// TwinCAT 3 PLC project Untitled1
// ProgramVersion: 3.1.4024.0
// libraries:
//   Tc2_Standard, * (Beckhoff Automation GmbH)
//   Tc2_System, * (Beckhoff Automation GmbH)
//   Tc3_Module, * (Beckhoff Automation GmbH)
// project tree:
//   DUTs/ KOMANDA.TcDUT, POZAYZ.TcDUT, POZICIJA.TcDUT, Valj.TcDUT
//   GVLs/ AUTO.TcGVL, GVL.TcGVL
//   / PlcTask.TcTTO
//   POUs/ AutoMove.TcPOU, Counter.TcPOU, Init.TcPOU, MAIN.TcPOU, Motor.TcPOU, MotorControla.TcPOU, Multiplex.TcPOU, Automatic.TcPOU, AutoMove2.TcPOU, Motor2.TcPOU, Test.TcPOU, TrackingLogic.TcPOU

CONFIGURATION Untitled1
    RESOURCE PLC ON TwinCAT3
        TASK PlcTask(INTERVAL := T#10ms, PRIORITY := 20);
        PROGRAM Automatic WITH PlcTask : Automatic;
    END_RESOURCE
END_CONFIGURATION

// ---- DUTs/KOMANDA.TcDUT
TYPE KOMANDA :
STRUCT
	I: INT;
	T: INT;
	P : INT;
END_STRUCT
END_TYPE

// ---- DUTs/POZAYZ.TcDUT
TYPE POZAYZ :
STRUCT
	A: INT;
	Y: INT;
	Z: INT;
END_STRUCT
END_TYPE

// ---- DUTs/POZICIJA.TcDUT
TYPE POZICIJA :
STRUCT
	A: INT;
	Y: INT;
	Z: INT;
	P: INT;
END_STRUCT
END_TYPE

// ---- DUTs/Valj.TcDUT
TYPE Valj :
STRUCT
	id: INT;
	pos: POZICIJA;
END_STRUCT
END_TYPE

// ---- GVLs/AUTO.TcGVL
{attribute 'qualified_only'}
VAR_GLOBAL
	Init : BOOL := FALSE;
	Varno :BOOL := FALSE;
	MotorIzbira : INT;
	VrtenjePremik : BOOL;
	VrtenjeSmer : BOOL;
	DvigPremik : BOOL;
	DvigSmer : BOOL;
	IztegPremik : BOOL;
	IztegSmer : BOOL;
	PrijemPremik : BOOL;
	PrijemSmer : BOOL;
	Current: POZICIJA;
	N: INT := 5; //v InstructionSize
	Komande0: ARRAY [0..4] OF POZICIJA := [(A := 0, Y := 0, Z := 0, P:= 0 ), 
		(A := 100, Y := 40, Z := 50, P:= 15 ),
		(A := 80, Y := 20, Z := 30, P:= 0 ),
		(A := 120, Y := 0, Z := 15, P:= 12 ),
		(A := 100, Y := 0, Z := 15, P:= 0 )];
	Status: INT := 0;
	PositionNum: INT := 2; // ne rabi
	ItemNumber : INT := 2; //ne rabi
	StageSelect : INT := 0;
	Recept : INT := 0;
	VRoki : INT := 0;
	Prijem : BOOL := FALSE;
	Positions: ARRAY [1..11] OF POZAYZ := [
			(A := 30, Y:=60, Z:= 105),
			(A := 30, Y:=60, Z:= 62),
			(A := 30, Y:=60, Z:= 20),
			(A := 60, Y:=60, Z:= 105),
			(A := 60, Y:=60, Z:= 62), // 5
			(A := 50, Y:=60, Z:= 105),
			(A := 50, Y:=60, Z:= 62),
			(A := 37, Y:=60, Z:= 105),
			(A := 40, Y:=45, Z:= 105),
			(A := 47, Y:=60, Z:= 105), // 10
			(A := 33, Y:=0, Z:= 50)];
	Items: ARRAY [1..5] OF POZAYZ := [
			(A := 5, Y:=60, Z:= 20),
			(A := 5, Y:=60, Z:= 62),
			(A := 5, Y:=60, Z:= 105),
			(A := 50, Y:=60, Z:= 105),
			(A := 50, Y:=60, Z:= 62)];
	StageMax : INT :=10;
	Stages :  ARRAY [1 .. 3] OF ARRAY [1 .. 9] OF KOMANDA :=  [[
		(I := 1, T := 0, P := 16),
		(I := 0, T := 1, P := 0),
		(I := 2, T := 0, P := 16),
		(I := 0, T := 2, P := 0),
		(I := 3, T := 0, P := 16), // 5
		(I := 0, T := 3, P := 0),
		(I := 2, T := 0, P := 16),
		(I := 0, T := 9, P := 0),
		(I := 0, T := 11, P := 0)],
[
		(I := 5, T := 0, P := 16),
		(I := 0, T := 4, P := 0),
		(I := 4, T := 0, P := 16),
		(I := 0, T := 5, P := 0),
		(I := 4, T := 0, P := 16), // 5
		(I := 0, T := 6, P := 0),
		(I := 5, T := 0, P := 16),
		(I := 0, T := 7, P := 0),
		(I := 0, T := 11, P := 0)],
[
		(I := 1, T := 0, P := 16),
		(I := 0, T := 10, P := 0),
		(I := 2, T := 0, P := 16),
		(I := 0, T := 8, P := 0),
		(I := 3, T := 0, P := 16), // 5
		(I := 0, T := 9, P := 0),
		(I := 3, T := 0, P := 16),
		(I := 0, T := 1, P := 0),
		(I := 0, T := 11, P := 0)]];
END_VAR

// ---- GVLs/GVL.TcGVL
{attribute 'Iualified_only'}


VAR_GLOBAL
	ToggleSwitch AT %I* : BOOL;
	LEDRed AT %Q* : BOOL;
	LEDGreen AT %Q* : BOOL;
	LEDUBlue AT %Q* : BOOL;
	LEDLBlue AT %Q* : BOOL;
	RedButton AT %I* : BOOL;
	GreenButton AT %I* : BOOL;
	ULBButton AT %I* : BOOL;
	URBButton AT %I* : BOOL;
	LLBButton AT %I* : BOOL;
	LRBButton AT %I* : BOOL;
	
	MVS AT %Q* : BOOL;
	MVP AT %Q* : BOOL;
	MIS AT %Q* : BOOL;
	MIP AT %Q* : BOOL;
	MDS AT %Q* : BOOL;
	MDP AT %Q* : BOOL;
	MPS AT %Q* : BOOL;
	MPP AT %Q* : BOOL;
	
	KSV AT %I* : BOOL;
	KSI AT %I* : BOOL;
	KSD AT %I* : BOOL;
	KSP AT %I* : BOOL;
	StV AT %I* : BOOL;
	StD AT %I* : BOOL;
	StI AT %I* : BOOL;
	StP AT %I* : BOOL;
END_VAR

// ---- POUs/Automatic.TcPOU
PROGRAM Automatic
VAR
	foo : BOOL;
	motor_1 : Motor2;
	auto_move : AutoMove;
	auto_move_2 : AutoMove2;
	tracking : TrackingLogic;
	init : Init;
END_VAR


init();
auto_move_2();
motor_1();
tracking();

END_PROGRAM

// ---- POUs/Motor2.TcPOU
FUNCTION_BLOCK Motor2
VAR_INPUT
END_VAR
VAR_OUTPUT
END_VAR
VAR
	sel1: BOOL := FALSE;
	sel2: BOOL := FALSE;
	sel3: BOOL := FALSE;
	sel4: BOOL := FALSE;
	mc1: motorControla;
	mc2: motorControla;
	mc3: motorControla;
	mc4: motorControla;
	interlock: BOOL;
	stop: BOOL;
END_VAR

IF GVL.ToggleSwitch = TRUE THEN
	AUTO.Varno := FALSE;
	IF GVL.ULBButton THEN
		sel1 := TRUE;
		sel2 := FALSE;
		sel3 := FALSE;
		sel4 := FALSE;
	ELSIF GVL.URBButton THEN
		sel1 := FALSE;
		sel2 := TRUE;
		sel3 := FALSE;
		sel4 := FALSE;
	ELSIF GVL.LLBButton THEN
		sel1 := FALSE;
		sel2 := FALSE;
		sel3 := TRUE;
		sel4 := FALSE;
	ELSIF GVL.LRBButton THEN
		sel1 := FALSE;
		sel2 := FALSE;
		sel3 := FALSE;
		sel4 := TRUE;
	END_IF
	
	mc1(		Premik := GVL.RedButton,
			Smer := GVL.GreenButton AND sel1,
			Select := sel1,
			KS := GVL.KSV,
			Step :=GVL.StV,
			Limes := 185,
			Position => AUTO.Current.A,
			OutSmer => GVL.MVS,
			OutPremik => GVL.MVP,
			Interlock => interlock,
			Stop => stop
			);
mc2(		Premik := GVL.RedButton,
			Smer := GVL.GreenButton AND sel2,
			Select := sel2,
			KS := GVL.KSD,
			Step :=GVL.StD,
			Limes := 105,
			Position => AUTO.Current.Z,
			OutSmer => GVL.MDS,
			OutPremik => GVL.MDP,
			Interlock => interlock,
			Stop => stop);
		mc3(
			Premik := GVL.RedButton,
			Smer := GVL.GreenButton AND sel3,
			Select := sel3,
			KS := GVL.KSI,
			Step :=GVL.StI,
			Limes := 65,
			Position => AUTO.Current.Y,
			OutSmer => GVL.MIS,
			OutPremik => GVL.MIP,
			Interlock => interlock,
			Stop => stop);
		mc4(
			Premik := GVL.RedButton,
			Smer := GVL.GreenButton AND sel4,
			Select := sel4,
			KS := GVL.KSP,
			Step :=GVL.StP,
			Limes := 16,
			Position => AUTO.Current.P,
			OutSmer => GVL.MPS,
			OutPremik => GVL.MPP,
			Interlock => interlock,
			Stop => stop);
ELSE
	CASE AUTO.MotorIzbira OF
		1:
		sel1 := TRUE;
		sel2 := FALSE;
		sel3 := FALSE;
		sel4 := FALSE;
	2:
		sel1 := FALSE;
		sel2 := TRUE;
		sel3 := FALSE;
		sel4 := FALSE;
	3:
		sel1 := FALSE;
		sel2 := FALSE;
		sel3 := TRUE;
		sel4 := FALSE;
	4:
		sel1 := FALSE;
		sel2 := FALSE;
		sel3 := FALSE;
		sel4 := TRUE;
	END_CASE
		mc1(
			Premik := AUTO.VrtenjePremik,
			Smer := AUTO.VrtenjeSmer,
			Select := sel1,
			KS := GVL.KSV,
			Step :=GVL.StV,
			Limes := 185,
			Position => AUTO.Current.A,
			OutPremik => GVL.MVP,
			OutSmer => GVL.MVS,
			Interlock => interlock,
			Stop => stop
			);
		mc2(
			Premik := AUTO.DvigPremik,
			Smer := AUTO.DvigSmer,
			Select := sel2,
			KS := GVL.KSD,
			Step :=GVL.StD,
			Limes := 105,
			Position => AUTO.Current.Z,
			OutPremik => GVL.MDP,
			OutSmer => GVL.MDS,
			Interlock => interlock,
			Stop => stop
			);
		
		IF AUTO.Current.Y = 0 AND AUTO.IztegSmer = TRUE THEN
			//GVL.LEDLBlue := TRUE;
			ELSE
			//.LEDLBlue := FALSE;
			mc3(
			Premik := AUTO.IztegPremik,
			Smer := AUTO.IztegSmer,
			Select := sel3,
			KS := GVL.KSI,
			Step :=GVL.StI,
			Limes := 60,
			Position => AUTO.Current.Y,
			OutPremik => GVL.MIP,
			OutSmer => GVL.MIS,
			Interlock => interlock,
			Stop => stop
			);
			END_IF
		mc4(
			Premik := AUTO.PrijemPremik,
			Smer := AUTO.PrijemSmer,
			Select := sel4,
			KS := GVL.KSP,
			Step :=GVL.StP,
			Limes := 16,
			Position => AUTO.Current.P,
			OutPremik => GVL.MPP,
			OutSmer => GVL.MPS,
			Interlock => interlock,
			Stop => stop
			);
END_IF

GVL.LEDGreen := stop;
GVL.LEDRed := interlock;

RETURN;

END_FUNCTION_BLOCK

// ---- POUs/MotorControla.TcPOU
FUNCTION_BLOCK MotorControla
VAR_INPUT
	Premik: BOOL;
	Smer: BOOL;
	Select: BOOL;
	KS: BOOL;
	Step: BOOL;
	Limes: WORD;
END_VAR
VAR_OUTPUT
	OutPremik: BOOL;
	OutSmer: BOOL;
	Interlock: BOOL;
	Stop: BOOL;
	Position: WORD;
END_VAR
VAR
	R_TRIG_0: R_TRIG;
	Dump: TIME;
	InL: TOF;
	RS_0: RS;

	R_TRIG_1: R_TRIG;
	TON0: TON;
	TON1: TON;
	TON_0: TON;
	Counter_0: Counter;
	F_TRIG_0: F_TRIG;
	InL1: TOF;
	IntL1: BOOL;
	IntL2: BOOL;
	IntL3: BOOL;
	R_TRIG_2: R_TRIG;
END_VAR
//dODAJ COLLISION DETECTION AND AVOIDANCE
//ZRIHTAJ SMER, KI SE SLABO SPREMINJA

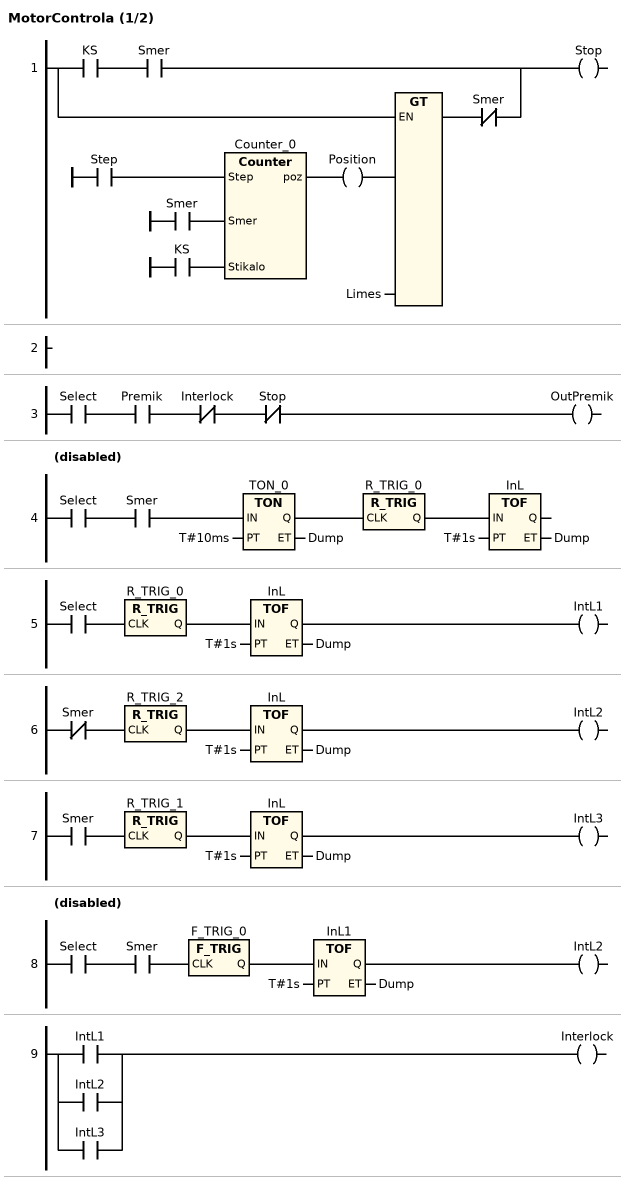
// NETWORK 1
Counter_0(Step := Step, Smer := Smer, Stikalo := KS); // Counter
Position := Counter_0.poz;
Stop := KS AND Smer OR Counter_0.poz > Limes AND NOT Smer;

// NETWORK 2

// NETWORK 3
OutPremik := Select AND Premik AND NOT Interlock AND NOT Stop;

// NETWORK 4 (disabled)
// TON_0(IN := Select AND Smer, PT := T#10ms, ET => Dump); // TON
// R_TRIG_0(CLK := TON_0.Q); // R_TRIG
// InL(IN := R_TRIG_0.Q, PT := T#1s, ET => Dump); // TOF

// NETWORK 5
R_TRIG_0(CLK := Select); // R_TRIG
InL(IN := R_TRIG_0.Q, PT := T#1s, ET => Dump); // TOF
IntL1 := InL.Q;

// NETWORK 6
R_TRIG_2(CLK := NOT Smer); // R_TRIG
InL(IN := R_TRIG_2.Q, PT := T#1s, ET => Dump); // TOF
IntL2 := InL.Q;

// NETWORK 7
R_TRIG_1(CLK := Smer); // R_TRIG
InL(IN := R_TRIG_1.Q, PT := T#1s, ET => Dump); // TOF
IntL3 := InL.Q;

// NETWORK 8 (disabled)
// F_TRIG_0(CLK := Select AND Smer); // F_TRIG
// InL1(IN := F_TRIG_0.Q, PT := T#1s, ET => Dump); // TOF
// IntL2 := InL1.Q;

// NETWORK 9
Interlock := IntL1 OR IntL2 OR IntL3;

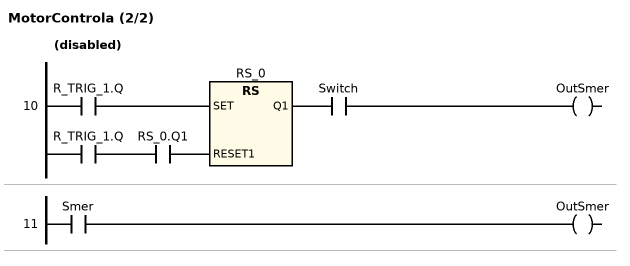
// NETWORK 10 (disabled)
// RS_0(SET := R_TRIG_1.Q, RESET1 := R_TRIG_1.Q AND RS_0.Q1); // RS
// OutSmer := RS_0.Q1 AND Switch;

// NETWORK 11
OutSmer := Smer;

END_FUNCTION_BLOCK

// ---- POUs/Counter.TcPOU
FUNCTION_BLOCK Counter
VAR_INPUT
	Step: BOOL;
	Smer: BOOL;
	Stikalo: BOOL;
END_VAR
VAR_OUTPUT
	poz: WORD;
END_VAR
VAR
	R_TRIG_0: R_TRIG;
	CTUD_0: Tc2_Standard.CTUD;
	R_TRIG_1: Tc2_Standard.R_TRIG;
END_VAR

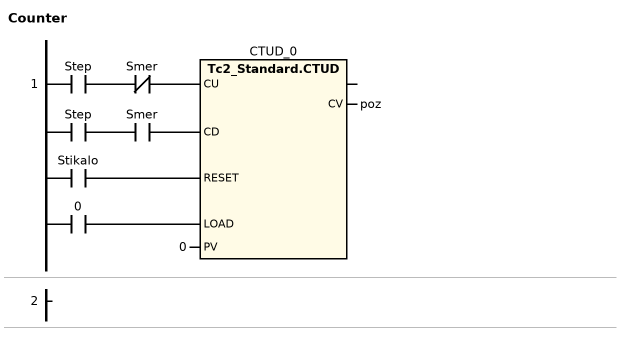
// NETWORK 1
CTUD_0(CU := Step AND NOT Smer, CD := Step AND Smer, RESET := Stikalo, LOAD := 0, PV := 0, CV => poz); // Tc2_Standard.CTUD

// NETWORK 2

END_FUNCTION_BLOCK

// ---- POUs/AutoMove.TcPOU
FUNCTION_BLOCK AutoMove
VAR_INPUT
END_VAR
VAR_OUTPUT
END_VAR
VAR
END_VAR

IF AUTO.Status > 0 AND AUTO.Status < AUTO.N THEN
	IF AUTO.Current.A <> AUTO.Komande0[AUTO.Status].A  THEN
		AUTO.MotorIzbira := 1;
		IF AUTO.Current.A > AUTO.Komande0[AUTO.Status].A THEN
			AUTO.VrtenjeSmer := TRUE;
		ELSE
			AUTO.VrtenjeSmer := FALSE;
		END_IF
		AUTO.VrtenjePremik := TRUE;
	ELSIF AUTO.Current.Y <> AUTO.Komande0[AUTO.Status].Y  THEN
		AUTO.MotorIzbira := 3;
		IF AUTO.Current.Y > AUTO.Komande0[AUTO.Status].Y THEN
			AUTO.IztegSmer := TRUE;
		ELSE
			AUTO.IztegSmer := FALSE;
		END_IF
		AUTO.IztegPremik := TRUE;
	ELSIF AUTO.Current.Z <> AUTO.Komande0[AUTO.Status].Z  THEN
		AUTO.MotorIzbira := 2;
		IF AUTO.Current.Z > AUTO.Komande0[AUTO.Status].Z THEN
			AUTO.DvigSmer := TRUE;
		ELSE
			AUTO.DvigSmer := FALSE;
		END_IF
		AUTO.DvigPremik := TRUE;
	ELSIF AUTO.Current.P <> AUTO.Komande0[AUTO.Status].P  THEN
		AUTO.MotorIzbira := 4;
		IF AUTO.Current.P > AUTO.Komande0[AUTO.Status].P THEN
			AUTO.PrijemSmer := TRUE;
		ELSE
			AUTO.PrijemSmer := FALSE;
		END_IF
		AUTO.PrijemPremik := TRUE;
	ELSE
		AUTO.VrtenjePremik := FALSE;
		AUTO.DvigPremik := FALSE;
		AUTO.IztegPremik := FALSE;
		AUTO.PrijemPremik := FALSE;
		AUTO.Status := AUTO.Status + 1;
	END_IF
END_IF

END_FUNCTION_BLOCK

// ---- POUs/AutoMove2.TcPOU
FUNCTION_BLOCK AutoMove2
VAR_INPUT
END_VAR
VAR_OUTPUT
END_VAR
VAR
	Target : POZAYZ;
END_VAR

IF AUTO.Init AND AUTO.StageSelect > 0 AND AUTO.StageSelect < AUTO.StageMax THEN
	IF AUTO.Varno = FALSE THEN
		AUTO.MotorIzbira := 3;
		AUTO.IztegSmer := TRUE;
		AUTO.IztegPremik := TRUE;
		IF AUTO.Current.Y = 0 THEN
			AUTO.Varno := TRUE;
		END_IF
	ELSIF AUTO.Stages[AUTO.Recept][Auto.StageSelect].I = 0 THEN
		Target := AUTO.Positions[AUTO.Stages[AUTO.Recept][Auto.StageSelect].T];
		IF AUTO.Current.Z <> Target.Z  THEN
			AUTO.MotorIzbira := 2;
			IF AUTO.Current.Z > Target.Z THEN
				AUTO.DvigSmer := TRUE;
			ELSE
				AUTO.DvigSmer := FALSE;
			END_IF
		AUTO.DvigPremik := TRUE;
		ELSIF AUTO.Current.A <> Target.A  THEN
			AUTO.MotorIzbira := 1;
			IF AUTO.Current.A > Target.A THEN
				AUTO.VrtenjeSmer := TRUE;
			ELSE
				AUTO.VrtenjeSmer := FALSE;
			END_IF
			AUTO.VrtenjePremik := TRUE;
		ELSIF AUTO.Current.Y <> Target.Y  THEN
			AUTO.MotorIzbira := 3;
			IF AUTO.Current.Y > Target.Y THEN
				AUTO.IztegSmer := TRUE;
			ELSE
				AUTO.IztegSmer := FALSE;
			END_IF
			AUTO.IztegPremik := TRUE;
		ELSIF AUTO.Current.P <> AUTO.Stages[AUTO.Recept][Auto.StageSelect].P  THEN
			AUTO.MotorIzbira := 4;
			IF AUTO.Current.P > AUTO.Stages[AUTO.Recept][Auto.StageSelect].P THEN
				AUTO.PrijemSmer := TRUE;
			ELSE
				AUTO.PrijemSmer := FALSE;
			END_IF
			AUTO.PrijemPremik := TRUE;
		ELSE
			AUTO.VrtenjePremik := FALSE;
			AUTO.DvigPremik := FALSE;
			AUTO.IztegPremik := FALSE;
			AUTO.PrijemPremik := FALSE;
			AUTO.StageSelect := AUTO.StageSelect + 1;
			AUTO.Varno := FALSE;
		END_IF
	ELSE
		Target := AUTO.Items[AUTO.Stages[AUTO.Recept][Auto.StageSelect].I];
			IF AUTO.Current.A <> Target.A  THEN
			AUTO.MotorIzbira := 1;
			IF AUTO.Current.A > Target.A THEN
				AUTO.VrtenjeSmer := TRUE;
			ELSE
				AUTO.VrtenjeSmer := FALSE;
			END_IF
			AUTO.VrtenjePremik := TRUE;
		ELSIF AUTO.Current.Z <> Target.Z  THEN
			AUTO.MotorIzbira := 2;
			IF AUTO.Current.Z > Target.Z THEN
				AUTO.DvigSmer := TRUE;
			ELSE
				AUTO.DvigSmer := FALSE;
			END_IF
			AUTO.DvigPremik := TRUE;
		ELSIF AUTO.Current.Y <> Target.Y  THEN
			AUTO.MotorIzbira := 3;
			IF AUTO.Current.Y > Target.Y THEN
				AUTO.IztegSmer := TRUE;
			ELSE
				AUTO.IztegSmer := FALSE;
			END_IF
			AUTO.IztegPremik := TRUE;
		ELSIF AUTO.Current.P <> AUTO.Stages[AUTO.Recept][Auto.StageSelect].P  THEN
			AUTO.MotorIzbira := 4;
			IF AUTO.Current.P > AUTO.Stages[AUTO.Recept][Auto.StageSelect].P THEN
				AUTO.PrijemSmer := TRUE;
			ELSE
				AUTO.PrijemSmer := FALSE;
			END_IF
			AUTO.PrijemPremik := TRUE;
		ELSE
			AUTO.VrtenjePremik := FALSE;
			AUTO.DvigPremik := FALSE;
			AUTO.IztegPremik := FALSE;
			AUTO.PrijemPremik := FALSE;
			AUTO.StageSelect := AUTO.StageSelect + 1;
			IF AUTO.StageSelect = AUTO.StageMax THEN
				AUTO.StageSelect := 0;
				AUTO.Init := FALSE;
				AUTO.Recept := 0;
			END_IF
			AUTO.Varno := FALSE;
		END_IF
	END_IF
	
END_IF

END_FUNCTION_BLOCK

// ---- POUs/Init.TcPOU
FUNCTION_BLOCK Init
VAR_INPUT
END_VAR
VAR_OUTPUT
END_VAR
VAR
END_VAR

IF NOT AUTO.Init AND GVL.ToggleSwitch = FALSE THEN
	IF NOT GVL.KSV THEN
		AUTO.MotorIzbira := 1;
		AUTO.VrtenjeSmer := TRUE;
		AUTO.VrtenjePremik := TRUE;
	ELSIF NOT GVL.KSD THEN
		AUTO.VrtenjePremik:= FALSE;
		AUTO.MotorIzbira := 2;
		AUTO.DvigSmer := TRUE;
		AUTO.DvigPremik := TRUE;
	ELSIF NOT GVL.KSP THEN
		AUTO.MotorIzbira := 4;
		AUTO.PrijemSmer := TRUE;
		AUTO.PrijemPremik := TRUE;
	ELSE
		AUTO.MotorIzbira := 0;
		AUTO.Current.Y := 0;
		IF GVL.ULBButton = TRUE THEN
			AUTO.Recept := 1;
		ELSIF GVL.URBButton = TRUE THEN
			AUTO.Recept:= 2;
		ELSIF GVL.LLBButton= TRUE THEN
			AUTO.Recept := 3;
		END_IF
		IF AUTO.Recept <> 0 THEN
			AUTO.StageSelect := 1;
			AUTO.Init := TRUE;
		END_IF
		
	END_IF
END_IF

END_FUNCTION_BLOCK

// ---- POUs/TrackingLogic.TcPOU
FUNCTION_BLOCK TrackingLogic
VAR_INPUT
END_VAR
VAR_OUTPUT
END_VAR
VAR
	target_ID : INT;
END_VAR

target_ID := AUTO.Stages[AUTO.Recept][AUTO.StageSelect].I;
IF AUTO.Current.P > 13 THEN
	AUTO.Prijem := TRUE;
ELSE
	AUTO.Prijem := FALSE;
END_IF
IF target_ID <> 0 AND AUTO.Current.P > 13 THEN
	AUTO.VRoki := target_ID;
	GVL.LEDLBlue := TRUE;
END_IF
IF AUTO.Current.P < 5 THEN
	AUTO.VRoki := 0;
	GVL.LEDLBlue := 0;
END_IF

IF AUTO.VRoki <> 0 THEN
	AUTO.Items[AUTO.VRoki].A := AUTO.Current.A;
	AUTO.Items[AUTO.VRoki].Y := AUTO.Current.Y;
	AUTO.Items[AUTO.VRoki].Z := AUTO.Current.Z; 
END_IF

END_FUNCTION_BLOCK

// ---- POUs/MAIN.TcPOU
PROGRAM MAIN
VAR
END_VAR

END_PROGRAM

// ---- POUs/Motor.TcPOU
FUNCTION_BLOCK Motor
VAR_INPUT
END_VAR
VAR_OUTPUT
END_VAR
VAR
	interlock : BOOL;
	stop: BOOL;
	motor_select : INT := 0;
	mc1 : MotorControla;
	mc2 : MotorControla;
	mc3 : MotorControla;
	mc4 : MotorControla;
	tst: BOOL := FALSE;
	dmp: WORD;
END_VAR

//manual control
GVL.MDP := FALSE;
GVL.MIP := FALSE;
GVL.MPP := FALSE;
GVL.MVP := FALSE;
IF GVL.ToggleSwitch = TRUE THEN
	AUTO.Varno := FALSE;
	IF GVL.ULBButton THEN
		motor_select := 1;
	ELSIF GVL.URBButton THEN
		motor_select := 2;
	ELSIF GVL.LLBButton THEN
		motor_select := 3;
	ELSIF GVL.LRBButton THEN
		motor_select := 4;
	END_IF
	
	CASE motor_select OF
		1: mc1(
			Premik := GVL.RedButton,
			Smer := GVL.GreenButton,
			Select := TRUE,
			KS := GVL.KSV,
			Step :=GVL.StV,
			Limes := 185,
			Position => AUTO.Current.A,
			OutSmer => GVL.MVS,
			OutPremik => GVL.MVP,
			Interlock => interlock,
			Stop => stop
			);
		2: mc2(
			Premik := GVL.RedButton,
			Smer := GVL.GreenButton,
			Select := TRUE,
			KS := GVL.KSD,
			Step :=GVL.StD,
			Limes := 105,
			Position => AUTO.Current.Z,
			OutSmer => GVL.MDS,
			OutPremik => GVL.MDP,
			Interlock => interlock,
			Stop => stop);
		3: mc3(
			Premik := GVL.RedButton,
			Smer := GVL.GreenButton,
			Select := TRUE,
			KS := GVL.KSI,
			Step :=GVL.StI,
			Limes := 65,
			Position => AUTO.Current.Y,
			OutSmer => GVL.MIS,
			OutPremik => GVL.MIP,
			Interlock => interlock,
			Stop => stop);
		4: mc4(
			Premik := GVL.RedButton,
			Smer := GVL.GreenButton,
			Select := TRUE,
			KS := GVL.KSP,
			Step :=GVL.StP,
			Limes := 16,
			Position => AUTO.Current.P,
			OutSmer => GVL.MPS,
			OutPremik => GVL.MPP,
			Interlock => interlock,
			Stop => stop);
	END_CASE
	
	GVL.LEDGreen := stop;
	GVL.LEDRed := interlock;
	
ELSE
	CASE AUTO.MotorIzbira OF
		1: mc1(
			Premik := AUTO.VrtenjePremik,
			Smer := AUTO.VrtenjeSmer,
			Select := TRUE,
			KS := GVL.KSV,
			Step :=GVL.StV,
			Limes := 185,
			Position => AUTO.Current.A,
			OutPremik => GVL.MVP,
			OutSmer => GVL.MVS,
			Interlock => interlock,
			Stop => stop
			);
		2: mc2(
			Premik := AUTO.DvigPremik,
			Smer := AUTO.DvigSmer,
			Select := TRUE,
			KS := GVL.KSD,
			Step :=GVL.StD,
			Limes := 105,
			Position => AUTO.Current.Z,
			OutPremik => GVL.MDP,
			OutSmer => GVL.MDS,
			Interlock => interlock,
			Stop => stop
			);
		
		3: IF AUTO.Current.Y = 0 AND AUTO.IztegSmer = TRUE THEN
			//GVL.LEDLBlue := TRUE;
			ELSE
			//.LEDLBlue := FALSE;
			mc3(
			Premik := AUTO.IztegPremik,
			Smer := AUTO.IztegSmer,
			Select := TRUE,
			KS := GVL.KSI,
			Step :=GVL.StI,
			Limes := 60,
			Position => AUTO.Current.Y,
			OutPremik => GVL.MIP,
			OutSmer => GVL.MIS,
			Interlock => interlock,
			Stop => stop
			);
			END_IF
		4: mc4(
			Premik := AUTO.PrijemPremik,
			Smer := AUTO.PrijemSmer,
			Select := TRUE,
			KS := GVL.KSP,
			Step :=GVL.StP,
			Limes := 16,
			Position => AUTO.Current.P,
			OutPremik => GVL.MPP,
			OutSmer => GVL.MPS,
			Interlock => interlock,
			Stop => stop
			);
	END_CASE
	
	GVL.LEDGreen := stop;
	GVL.LEDRed := interlock;
	
END_IF

RETURN;

END_FUNCTION_BLOCK

// ---- POUs/Multiplex.TcPOU
FUNCTION_BLOCK Multiplex
VAR_INPUT
	In1: BOOL;
	In2: BOOL;
	In3: BOOL;
END_VAR
VAR_OUTPUT
	Out1: BOOL;
	Out2: BOOL;
	Out3: BOOL;
	Out4: BOOL;
END_VAR
VAR
	RS_1: RS;
	RS_2: RS;
	RS_3: RS;
	RS_5: RS;
	TON_4: TON;
	TON_3: TON;
	TON_2: TON;
	TON_1: TON;
END_VAR

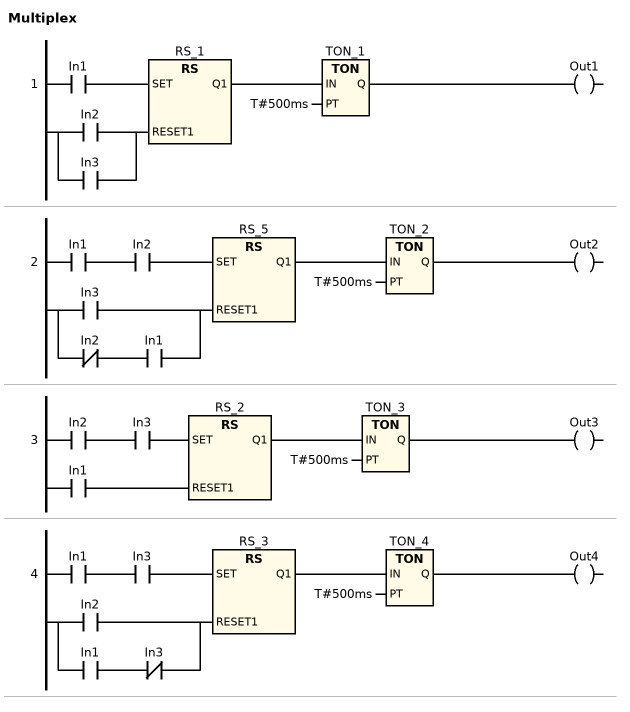
// NETWORK 1
RS_1(SET := In1, RESET1 := In2 OR In3); // RS
TON_1(IN := RS_1.Q1, PT := T#500ms); // TON
Out1 := TON_1.Q;

// NETWORK 2
RS_5(SET := In1 AND In2, RESET1 := In3 OR NOT In2 AND In1); // RS
TON_2(IN := RS_5.Q1, PT := T#500ms); // TON
Out2 := TON_2.Q;

// NETWORK 3
RS_2(SET := In2 AND In3, RESET1 := In1); // RS
TON_3(IN := RS_2.Q1, PT := T#500ms); // TON
Out3 := TON_3.Q;

// NETWORK 4
RS_3(SET := In1 AND In3, RESET1 := In2 OR In1 AND NOT In3); // RS
TON_4(IN := RS_3.Q1, PT := T#500ms); // TON
Out4 := TON_4.Q;

END_FUNCTION_BLOCK

// ---- POUs/Test.TcPOU
PROGRAM Test
VAR
	EdgeD: R_TRIG;
	RS_0: RS;
	CTU_0: CTUD;
	COUNT: CTUD;
	testVar1 : WORD := 11;
	testVar2 : WORD := 0;
	testVar3 : WORD := 12;
		testVar4 : BOOL := TRUE;
		TP_0: TP;
	testVar5 : TIME := T#0ms;
	LEDUBlue: BOOL;
	ms: TIME;
	T1: TON;
	TOF_0: TOF;
	LLBButton: BOOL;
	LED: MotorControla;
	MotorControla_0: MotorControla;
	MotorControla_1: MotorControla;
	MotorControla_2: MotorControla;
	MX: Multiplex;
	Patch: MotorControla;
	MotorControla_3: MotorControla;
	MotorControla_4: MotorControla;
	MotorControla_5: MotorControla;
	IntLck: BOOL;
	IntLck1: BOOL;
	IntLck2: BOOL;
	IntLck3: BOOL;
	Stp3: BOOL;
	Stp1: BOOL;
	Stp2: BOOL;
	Stp4: BOOL;
	Counter_0: Counter;
	KDP: BOOL;
	IntLck4: BOOL;
END_VAR

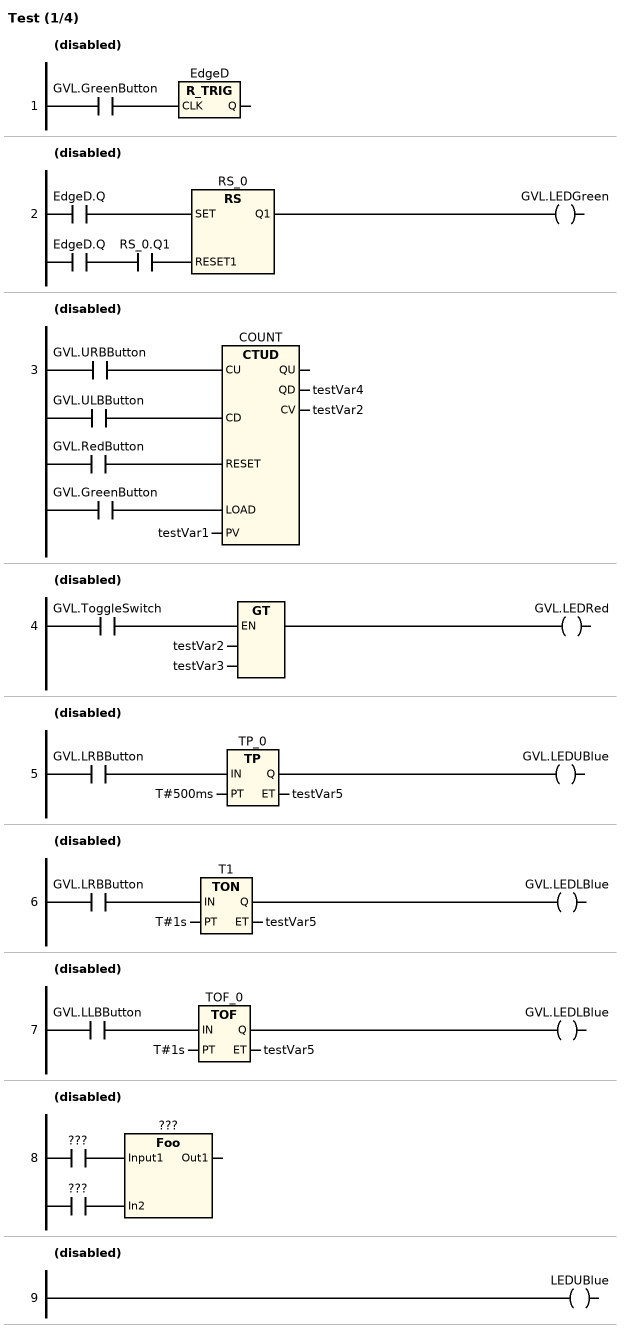
// NETWORK 1 (disabled)
// EdgeD(CLK := GVL.GreenButton); // R_TRIG

// NETWORK 2 (disabled)
// RS_0(SET := EdgeD.Q, RESET1 := EdgeD.Q AND RS_0.Q1); // RS
// GVL.LEDGreen := RS_0.Q1;

// NETWORK 3 (disabled)
// COUNT(
//     CU := GVL.URBButton,
//     CD := GVL.ULBButton,
//     RESET := GVL.RedButton,
//     LOAD := GVL.GreenButton,
//     PV := testVar1,
//     QD => testVar4,
//     CV => testVar2); // CTUD

// NETWORK 4 (disabled)
// GVL.LEDRed := GVL.ToggleSwitch AND testVar2 > testVar3;

// NETWORK 5 (disabled)
// TP_0(IN := GVL.LRBButton, PT := T#500ms, ET => testVar5); // TP
// GVL.LEDUBlue := TP_0.Q;

// NETWORK 6 (disabled)
// T1(IN := GVL.LRBButton, PT := T#1s, ET => testVar5); // TON
// GVL.LEDLBlue := T1.Q;

// NETWORK 7 (disabled)
// TOF_0(IN := GVL.LLBButton, PT := T#1s, ET => testVar5); // TOF
// GVL.LEDLBlue := TOF_0.Q;

// NETWORK 8 (disabled)
// ???(); // Foo

// NETWORK 9 (disabled)
// LEDUBlue := TRUE;

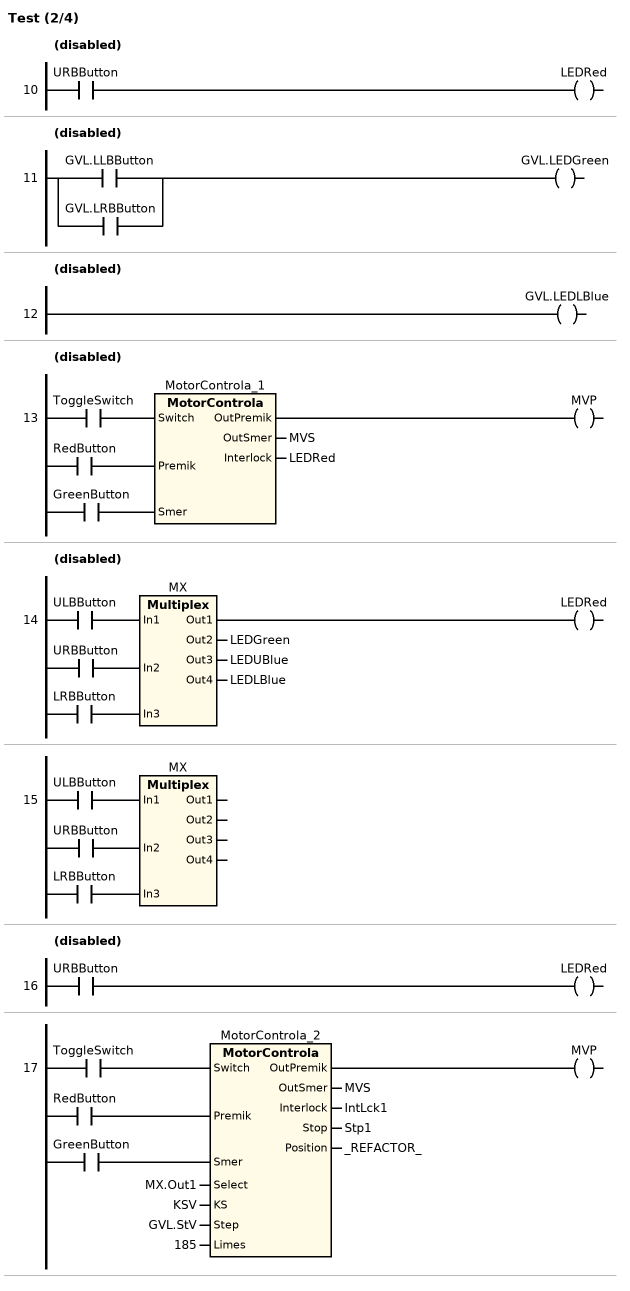
// NETWORK 10 (disabled)
// LEDRed := URBButton;

// NETWORK 11 (disabled)
// GVL.LEDGreen := GVL.LLBButton OR GVL.LRBButton;

// NETWORK 12 (disabled)
// GVL.LEDLBlue := TRUE;

// NETWORK 13 (disabled)
// MotorControla_1(
//     Switch := ToggleSwitch,
//     Premik := RedButton,
//     Smer := GreenButton,
//     OutSmer => MVS,
//     Interlock => LEDRed); // MotorControla
// MVP := MotorControla_1.OutPremik;

// NETWORK 14 (disabled)
// MX(
//     In1 := ULBButton,
//     In2 := URBButton,
//     In3 := LRBButton,
//     Out2 => LEDGreen,
//     Out3 => LEDUBlue,
//     Out4 => LEDLBlue); // Multiplex
// LEDRed := MX.Out1;

// NETWORK 15
MX(In1 := ULBButton, In2 := URBButton, In3 := LRBButton); // Multiplex

// NETWORK 16 (disabled)
// LEDRed := URBButton;

// NETWORK 17
MotorControla_2(
    Switch := ToggleSwitch,
    Premik := RedButton,
    Smer := GreenButton,
    Select := MX.Out1,
    KS := KSV,
    Step := GVL.StV,
    Limes := 185,
    OutSmer => MVS,
    Interlock => IntLck1,
    Stop => Stp1,
    Position => _REFACTOR_); // MotorControla
MVP := MotorControla_2.OutPremik;

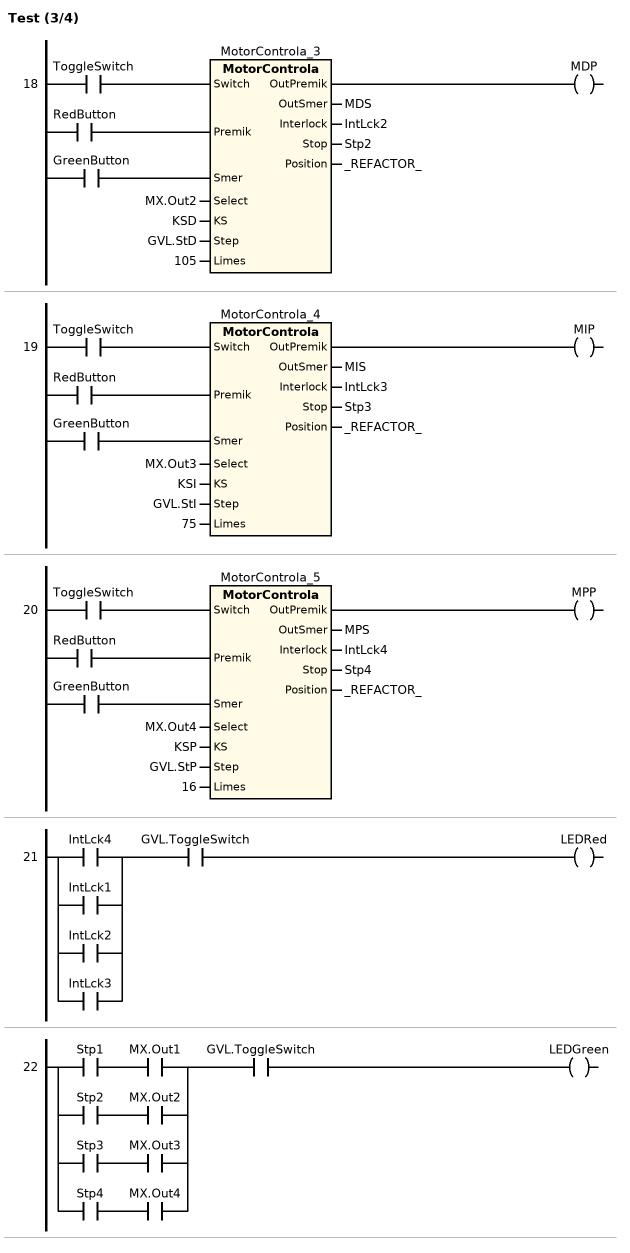
// NETWORK 18
MotorControla_3(
    Switch := ToggleSwitch,
    Premik := RedButton,
    Smer := GreenButton,
    Select := MX.Out2,
    KS := KSD,
    Step := GVL.StD,
    Limes := 105,
    OutSmer => MDS,
    Interlock => IntLck2,
    Stop => Stp2,
    Position => _REFACTOR_); // MotorControla
MDP := MotorControla_3.OutPremik;

// NETWORK 19
MotorControla_4(
    Switch := ToggleSwitch,
    Premik := RedButton,
    Smer := GreenButton,
    Select := MX.Out3,
    KS := KSI,
    Step := GVL.StI,
    Limes := 75,
    OutSmer => MIS,
    Interlock => IntLck3,
    Stop => Stp3,
    Position => _REFACTOR_); // MotorControla
MIP := MotorControla_4.OutPremik;

// NETWORK 20
MotorControla_5(
    Switch := ToggleSwitch,
    Premik := RedButton,
    Smer := GreenButton,
    Select := MX.Out4,
    KS := KSP,
    Step := GVL.StP,
    Limes := 16,
    OutSmer => MPS,
    Interlock => IntLck4,
    Stop => Stp4,
    Position => _REFACTOR_); // MotorControla
MPP := MotorControla_5.OutPremik;

// NETWORK 21
LEDRed := (IntLck4 OR IntLck1 OR IntLck2 OR IntLck3) AND GVL.ToggleSwitch;

// NETWORK 22
LEDGreen := (Stp1 AND MX.Out1 OR Stp2 AND MX.Out2 OR Stp3 AND MX.Out3 OR Stp4 AND MX.Out4) AND GVL.ToggleSwitch;

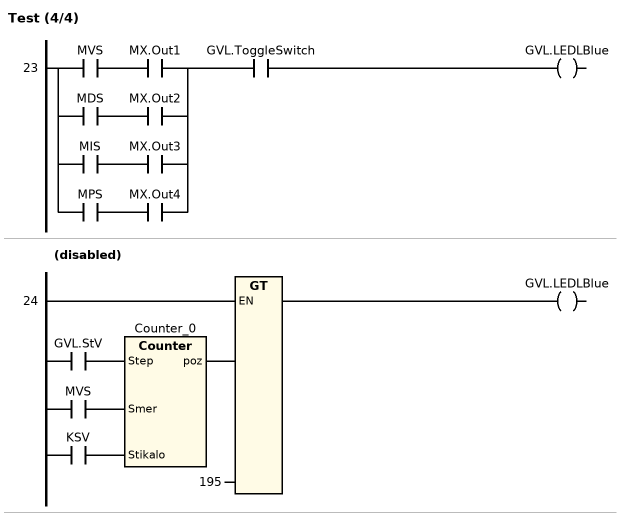
// NETWORK 23
GVL.LEDLBlue := (MVS AND MX.Out1 OR MDS AND MX.Out2 OR MIS AND MX.Out3 OR MPS AND MX.Out4) AND GVL.ToggleSwitch;

// NETWORK 24 (disabled)
// Counter_0(Step := GVL.StV, Smer := MVS, Stikalo := KSV); // Counter
// GVL.LEDLBlue := Counter_0.poz > 195;

END_PROGRAM
